Fanuc KAREL source: IO0202.KL

PROGRAM IO0202
%STACKSIZE=65535
%PRIORITY=65535
%NOLOCKGROUP
ROUTINE RTEST FROM IO0202
ROUTINE RTEST
VAR
L1 : ARRAY[3] OF INTEGER
L2 : XYZWPR
L3 : JOINTPOS9
L4 : POSITION
U2C_37 : BOOLEAN -- ASSUMED 2C source type; see uncertainty report
S1 : INTEGER
U2C_39 : REAL -- ASSUMED 2C source type; see uncertainty report
U2C_40 : BOOLEAN -- ASSUMED 2C source type; see uncertainty report
U2C_41 : INTEGER -- ASSUMED 2C source type; see uncertainty report
BEGIN
U2C_37=TRUE
L1[1]=2
U2C_40=TRUE
U2C_41=1065353216
-- UNSAFE_SOURCE_IR line 20: SET_EPOS_REG(1, convert_xyzwpr_to_xyzwprext(L2), S1, 1)
END RTEST
BEGIN
RTEST
END IO0202
